FUNCTION_BLOCK AtvResetError (* Composite Function Block Type *)
  (* Standard: 61499-2 *)
  (* Version 0.0, 8/19/2024, SESA713705, Schneider Electric, template *)
  PACKAGE SE.Nereda;
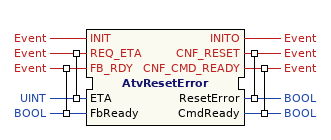
  EVENT_INPUT
    INIT; (* Initializes the symbolic link data destination FB with N (1 <= N <= 16) variables *)
    REQ_ETA WITH ETA; (* Normal Execution Request *)
    FB_RDY WITH FbReady;
  END_EVENT
  EVENT_OUTPUT
    INITO; (* Initialization confirm *)
    CNF_RESET WITH ResetError; (* Execution Confirmation *)
    CNF_CMD_READY WITH CmdReady;
  END_EVENT
  VAR_INPUT
    ETA : UINT;
    FbReady : BOOL;
  END_VAR
  VAR_OUTPUT
    ResetError : BOOL;
    CmdReady : BOOL;
  END_VAR
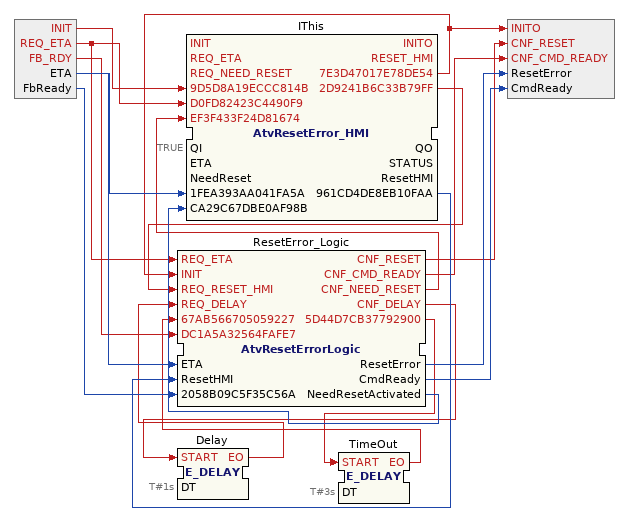
  (* 06 - HMI INTERFACE *)
  (* 02 - FUNCTIONNAL OUTPUT INTERFACE *)
  (* 05 - LOGIC *)
  (* 01 - FUNCTIONNAL INPUT INTERFACE *)
  FBS
    IThis : AtvResetError_HMI(QI := TRUE);
    ResetError_Logic : AtvResetErrorLogic;
    Delay : E_DELAY(DT := T#1s);
    TimeOut : E_DELAY(DT := T#3s);
  END_FBS
  EVENT_CONNECTIONS
    REQ_ETA TO ResetError_Logic.REQ_ETA;
    ResetError_Logic.CNF_RESET TO CNF_RESET;
    ResetError_Logic.CNF_CMD_READY TO CNF_CMD_READY;
    INIT TO IThis.9D5D8A19ECCC814B;
    REQ_ETA TO IThis.D0FD82423C4490F9;
    ResetError_Logic.CNF_NEED_RESET TO IThis.EF3F433F24D81674;
    IThis.7E3D47017E78DE54 TO INITO;
    IThis.7E3D47017E78DE54 TO ResetError_Logic.INIT;
    IThis.2D9241B6C33B79FF TO ResetError_Logic.REQ_RESET_HMI;
    ResetError_Logic.CNF_DELAY TO Delay.START;
    Delay.EO TO ResetError_Logic.REQ_DELAY;
    ResetError_Logic.5D44D7CB37792900 TO TimeOut.START;
    TimeOut.EO TO ResetError_Logic.67AB566705059227;
    FB_RDY TO ResetError_Logic.DC1A5A32564FAFE7;
  END_CONNECTIONS
  DATA_CONNECTIONS
    ETA TO ResetError_Logic.ETA;
    ResetError_Logic.ResetError TO ResetError;
    ResetError_Logic.CmdReady TO CmdReady;
    ETA TO IThis.1FEA393AA041FA5A;
    ResetError_Logic.NeedResetActivated TO IThis.CA29C67DBE0AF98B;
    IThis.961CD4DE8EB10FAA TO ResetError_Logic.ResetHMI;
    FbReady TO ResetError_Logic.2058B09C5F35C56A;
  END_CONNECTIONS
END_FUNCTION_BLOCK
